Yaskawa INFORM job: R1_W63-A1(120,-90)KM-OK.JBI

/JOB
//NAME R1_W63-A1(120,-90)KM-OK
///FOLDERNAME KRIS-SCIANA
//POS
///NPOS 37,37,0,3,0,0
///TOOL 0
///POSTYPE PULSE
///PULSE
C00000=21526,-168629,-93491,-40042,64194,-11475
C00001=50807,-130476,-89227,-36607,58876,-89355
C00002=109362,-75319,-65328,-35955,92155,-75859
C00003=124724,-69895,-47330,-35587,95301,-70457
C00004=122746,-71974,-45016,-35776,92438,-70340
C00005=121897,-70613,-41698,-35873,90988,-70217
C00006=121906,-70690,-40639,-35855,90422,-70032
C00007=121912,-71656,-41849,-35857,90631,-70092
C00008=121929,-72977,-42409,-35846,90363,-69999
C00009=121912,-71656,-41849,-35857,90631,-70092
C00010=120115,-70592,-41831,-36173,90325,-70724
C00011=118643,-70559,-41816,-36411,89716,-71125
C00012=120115,-70592,-41831,-36173,90325,-70724
C00013=120458,-70126,-43591,-36160,91548,-70986
C00014=122490,-68131,-45927,-35960,94406,-71089
C00015=120040,-69244,-55307,-16934,100757,-64886
C00016=144710,-62962,-53793,4762,102395,-56460
C00017=146144,-67957,-53971,4977,99861,-56060
C00018=145832,-65988,-49619,4892,98219,-56232
C00019=145912,-65817,-48327,4898,97509,-56235
C00020=145912,-66142,-49216,4904,97888,-56220
C00021=146397,-68232,-50171,4985,97375,-56074
C00022=146112,-67098,-49850,4939,97776,-56156
C00023=115509,-75384,-45500,33781,91615,-70126
C00024=116402,-75454,-45530,33942,91251,-69881
C00025=112362,-75031,-45344,33188,92909,-70988
C00026=118570,-49874,-41855,6042,115556,21537
C00027=120548,-60633,-53702,-6492,107288,80293
C00028=112885,-79464,-55237,-10195,90684,79138
C00029=120580,-32197,-17712,-5125,118654,79669
C00030=120572,-32853,-19191,-5161,119225,79639
C00031=133182,-79168,-55625,8207,90817,85074
C00032=133565,-79462,-55970,8253,90839,85204
C00033=113854,-76943,-50277,22812,92897,77520
C00034=104672,-74688,-61326,16011,101183,75838
C00035=70152,-153187,-124769,8200,55972,64027
C00036=22999,-153190,-124770,8193,30097,64033
BC00000=122859,1188774,1068222
BC00001=56396,1189606,1068222
BC00002=93202,1189606,1068222
BC00003=127572,1189606,1068222
BC00004=127572,1189606,1068222
BC00005=127572,1189606,1068222
BC00006=127572,1189606,1068222
BC00007=127572,1189606,1068222
BC00008=127572,1189606,1068222
BC00009=127572,1189606,1068222
BC00010=127572,1189606,1068222
BC00011=127572,1189606,1068222
BC00012=127572,1189606,1068222
BC00013=127572,1189606,1068222
BC00014=127572,1189606,1068222
BC00015=121474,1189606,1068222
BC00016=121474,1189606,1068222
BC00017=121474,1189606,1068222
BC00018=121474,1189606,1068222
BC00019=121474,1189606,1068222
BC00020=121474,1189606,1068222
BC00021=121474,1189606,1068222
BC00022=121474,1189606,1068222
BC00023=121474,1189606,1068222
BC00024=121474,1189606,1068222
BC00025=121474,1189606,1068222
BC00026=133718,1189606,1068222
BC00027=152672,1189606,1068222
BC00028=161950,1189606,1068221
BC00029=153597,1189606,1068222
BC00030=153597,1189606,1068222
BC00031=161951,1189606,1068222
BC00032=101567,1189606,1068222
BC00033=96797,1189605,1068221
BC00034=94818,1189606,1068222
BC00035=94818,1189606,1068222
BC00036=94818,1158137,1068222
///POSTYPE BASE
///RECTAN
///RCONF 0,0,0,0,0,0,0,0,0,0,0,0,0,0,0,0,0,0,0,0,0,0,0,0
P00006=0.222,-3.123,-1.508,0.0000,0.0000,0.0000
P00021=-0.225,-6.128,-0.405,0.0000,0.0000,0.0000
P00022=0.222,-3.123,-1.508,0.0000,0.0000,0.0000
//INST
///DATE 2024/07/25 17:49
///ATTR SC,RW
///GROUP1 RB1,BS1
NOP
'r1_W63-A1(120,-90)
'Path S1498
SFTOF
MOVJ C00000 BC00000 VJ=20.00
MOVJ C00001 BC00001 VJ=20.00
MOVJ C00002 BC00002 VJ=20.00
MOVJ C00003 BC00003 VJ=20.00
MOVJ C00004 BC00004 VJ=20.00
MOVL C00005 BC00005 V=60.0
REFP 3 C00006 BC00006
CALL JOB:SEARCH-R1
SET P021 P006
SFTON P021
MOVL C00007 BC00007 V=60.0
REFP 3 C00008 BC00008
CALL JOB:SEARCH-R1
SET P021 P006
SFTON P021
MOVL C00009 BC00009 V=60.0
MOVL C00010 BC00010 V=60.0
REFP 3 C00011 BC00011
CALL JOB:SEARCH-R1
SET P021 P006
SFTON P021
MOVL C00012 BC00012 V=60.0
MOVL C00013 BC00013 V=100.0
MOVL C00014 BC00014 V=166.7
'Path S1499
SFTOF
MOVJ C00015 BC00015 VJ=20.00
MOVJ C00016 BC00016 VJ=20.00
MOVJ C00017 BC00017 VJ=20.00
MOVL C00018 BC00018 V=166.7
REFP 3 C00019 BC00019
CALL JOB:SEARCH-R1
SET P022 P006
SFTON P022
MOVL C00020 BC00020 V=60.0
REFP 3 C00021 BC00021
CALL JOB:SEARCH-R1
SET P022 P006
SFTON P022
MOVL C00022 BC00022 V=60.0
MOVL C00023 BC00023 V=166.7
REFP 3 C00024 BC00024
CALL JOB:SEARCH-R1
SET P022 P006
MOVL C00025 BC00025 V=250.0
SFTON P022
'Path W1500
SFTOF
SFTON P022
MOVJ C00026 BC00026 VJ=20.00
MOVJ C00027 BC00027 VJ=20.00
SFTON P021
MOVL C00028 BC00028 V=100.0 PL=0
REFP 1 C00029 BC00029
REFP 2 C00030 BC00030
MACRO1 MJ#(0) ARGF7
ARCON
MOVL C00031 BC00031 V=11.2
SFTON P022
MOVL C00032 BC00032 V=11.2
SFTON P022
MOVL C00033 BC00033 V=11.2
ARCOF
SFTOF
MOVL C00034 BC00034 V=250.0
MOVL C00035 BC00035 V=666.7
MOVJ C00036 BC00036 VJ=20.00
SFTOF
END
